FUNCTION_BLOCK File IMPLEMENTS Cyclic
VAR
	_Busy : BOOL;
	_Done : BOOL;
	_Error : BOOL;
	
	openRequest : BOOL;
	readRequest : BOOL;
	writeRequest : BOOL;
	appendMode : BOOL;
	filePath : T_MaxString;
	
	buffer : POINTER TO BYTE;
	bufferLength : UDINT;

	handle : UINT;
	opener : FB_FileOpen;
	closer : FB_FileClose;
	reader : FB_FileRead;
	writer : FB_FileWrite;
	
	fileState : (Waiting, OpenMode, Opening, Reading, Writing, Closing);
	
	filenameForAlarm : T_MaxString;
	openErrorTrigger : R_TRIG;
	readErrorTrigger : R_TRIG;
	writeErrorTrigger : R_TRIG;
	closeErrorTrigger : R_TRIG;
	notFoundError : MessageEventLogger(TC_EVENTS.FileEventClass.InvalidPath);
	fileOpenError : MessageEventLogger(TC_EVENTS.FileEventClass.OpenFileError);
	fileReadError : MessageEventLogger(TC_EVENTS.FileEventClass.ReadFileError);
	fileWriteError : MessageEventLogger(TC_EVENTS.FileEventClass.WriteFileError);
	fileCloseError : MessageEventLogger(TC_EVENTS.FileEventClass.CloseFileError);
END_VAR
VAR CONSTANT
	NotFoundErrorNumber : UDINT := 16#70C;
END_VAR

{attribute 'monitoring' := 'call'}
PROPERTY Busy : BOOL
GET
Busy := _Busy;
END_GET
END_PROPERTY

METHOD Cyclic
CASE fileState OF
	
	Waiting:
	
		IF (openRequest) THEN
			openRequest := FALSE;
			_Done := FALSE;
			
			fileState := OpenMode;
		END_IF
	
	OpenMode:
	
		IF (readRequest) THEN
			opener.nMode := FOPEN_MODEREAD;
		ELSIF (writeRequest) THEN
			IF (appendMode) THEN
				opener.nMode := FOPEN_MODEAPPEND;
			ELSE
				opener.nMode := FOPEN_MODEWRITE;
			END_IF
		END_IF
		
		opener.nMode := opener.nMode OR FOPEN_MODETEXT;

		fileState := Opening;
	
	Opening:
	
		opener(
			bExecute := NOT opener.bBusy,
			sPathName := filePath,
			hFile => handle,
		);
		
		IF (NOT opener.bExecute AND NOT opener.bBusy AND handle <> 0) THEN
			opener();
			IF (readRequest) THEN
				fileState := Reading;
			ELSIF (writeRequest) THEN
				fileState := Writing;
			END_IF
		END_IF
	
	Reading:
	
		reader(
			bExecute := NOT reader.bBusy,
			hFile := handle,
			pReadBuff := buffer,
			cbReadLen := bufferLength,
		);
		
		IF (NOT reader.bExecute AND NOT reader.bBusy) THEN
			fileState := Closing;
		END_IF
	
	Writing:
	
		writer(
			bExecute := NOT writer.bBusy,
			hFile := handle,
			pWriteBuff := buffer,
			cbWriteLen := bufferLength,
		);
		
		IF (NOT writer.bExecute AND NOT writer.bBusy) THEN
			fileState := Closing;
		END_IF
	
	Closing:
	
		IF (handle = 0) THEN
			fileState := Waiting;
		ELSE
			closer(
				bExecute := NOT closer.bBusy,
				hFile := handle,
			);
			
			IF (NOT closer.bExecute AND NOT closer.bBusy) THEN
				closer();
				handle := 0;
				_Done := TRUE;
				
				fileState := Waiting;
			END_IF
		END_IF
	
END_CASE

_Busy := fileState <> Waiting;

openErrorTrigger(CLK := opener.bError);
readErrorTrigger(CLK := reader.bError);
writeErrorTrigger(CLK := writer.bError);
closeErrorTrigger(CLK := closer.bError);
_Error := 
	openErrorTrigger.Q
	OR readErrorTrigger.Q
	OR writeErrorTrigger.Q
	OR closeErrorTrigger.Q
	;
IF (_Error) THEN
	openRequest := FALSE;
	readRequest := FALSE;
	writeRequest := FALSE;
	
	filenameForAlarm := opener.sPathName;
	IF (EventParameters.EscapeBackslash) THEN
		filenameForAlarm := ReplaceAll(filenameForAlarm, '\', '\\'); // Escape backslash to use with web-based HMIs
	END_IF
	
	IF (openErrorTrigger.Q AND opener.nErrId = NotFoundErrorNumber) THEN
		notFoundError.Arguments.Clear().AddStringByValue(filenameForAlarm);
		notFoundError.Send();
	ELSIF (openErrorTrigger.Q) THEN
		fileOpenError.Arguments.Clear().AddStringByValue(filenameForAlarm);
		fileOpenError.Send();
	ELSIF (readErrorTrigger.Q) THEN
		fileReadError.Arguments.Clear().AddStringByValue(filenameForAlarm);
		fileReadError.Send();
	ELSIF (openErrorTrigger.Q) THEN
		fileWriteError.Arguments.Clear().AddStringByValue(filenameForAlarm);
		fileWriteError.Send();
	ELSIF (openErrorTrigger.Q) THEN
		fileCloseError.Arguments.Clear().AddStringByValue(filenameForAlarm);
		fileCloseError.Send();
	END_IF
	
	IF (fileState > Waiting AND fileState < Closing) THEN
		fileState := Closing;
	END_IF
END_IF
END_METHOD

{attribute 'monitoring' := 'call'}
PROPERTY Done : BOOL
GET
Done := _Done;
END_GET
END_PROPERTY

{attribute 'monitoring' := 'call'}
PROPERTY Error : BOOL
GET
Error := _Error;
END_GET
END_PROPERTY

METHOD Read
VAR_INPUT
	buffer : POINTER TO BYTE;
	bufferLength : UDINT;
	filePath : T_MaxString;
END_VAR
IF (NOT _Busy) THEN
	THIS^.filePath := filePath;
	THIS^.buffer := buffer;
	THIS^.bufferLength := bufferLength;
	
	openRequest := TRUE;
	readRequest := TRUE;
	writeRequest := FALSE;
END_IF
END_METHOD

METHOD Write
VAR_INPUT
	buffer : POINTER TO BYTE;
	bufferLength : UDINT;
	filePath : T_MaxString;
	append : BOOL;
END_VAR
IF (NOT _Busy) THEN
	THIS^.filePath := filePath;
	THIS^.buffer := buffer;
	THIS^.bufferLength := bufferLength;
	
	openRequest := TRUE;
	writeRequest := TRUE;
	readRequest := FALSE;
	appendMode := append;
END_IF
END_METHOD

END_FUNCTION_BLOCK

(* stored: Version 1.1.0.1
   POU File: Id {de1840e6-6126-0b1b-3259-f1ec0dc2154b}, SpecialFunc None
   Property Busy: Id {39637069-ad71-0e7b-2708-deacacfec070}
   Get Get: Id {101c984c-f4d0-0197-2073-acf04044788f}
   Method Cyclic: Id {d7851b7e-e8df-0535-3f15-3ce94d3bda28}
   Property Done: Id {55291a61-d05b-0a48-3c18-6798884dc6b1}
   Get Get: Id {b8c8defc-19ee-0f08-37b2-31b3ca24ac43}
   Property Error: Id {2b9e7ff5-57e3-0de2-1849-56ea242c89c0}
   Get Get: Id {84d83e28-8398-0028-3541-5cbea1ee2adb}
   Method Read: Id {864f7368-a611-0ae8-28b2-0d3f9d414814}
   Method Write: Id {b6e90204-5ab5-0a36-123e-8ee0b5b32492} *)
